// TIA Portal V18 export
// export: Created 2025-12-01T17:50:25.5329031Z, ExportSetting None, DisplayName Totally Integrated Automation Portal, DisplayVersion V18 Update 5, DisplayName TIA Portal Openness, DisplayVersion V18 Update 5, DisplayName TIA Portal Teamcenter Gateway, DisplayVersion V18, DisplayName TIA Portal Version Control Interface, DisplayVersion V18, DisplayName STEP 7 Professional, DisplayVersion V18 Update 5, DisplayName STEP 7 Safety, DisplayVersion V18, DisplayName WinCC Professional, DisplayVersion V18 Update 5
ORGANIZATION_BLOCK "07_CYCL_FLT"   // OB80, STL, TimeErrorInterrupt
TITLE = "Cycle Time Fault"
{ S7_Optimized_Access := 'FALSE' }
   VAR_TEMP
      OB80_EV_CLASS : Byte;   // 16#35, Event class 3, Entering event state, Internal fault event
      OB80_FLT_ID : Byte;   // 16#XX, Fault identifcation code
      OB80_PRIORITY : Byte;   // Priority of OB Execution
      OB80_OB_NUMBR : Byte;   // 80 (Organization block 80, OB80)
      OB80_RESERVED_1 : Byte;   // Reserved for system
      OB80_RESERVED_2 : Byte;   // Reserved for system
      OB80_ERROR_INFO : Word;   // Error information on event
      OB80_ERR_EV_CLASS : Byte;   // Class of event causing error
      OB80_ERR_EV_NUM : Byte;   // Number of event causing error
      OB80_OB_PRIORITY : Byte;   // Priority of OB causing error
      OB80_OB_NUM : Byte;   // Number of OB causing error
      OB80_DATE_TIME : Date_And_Time;   // Date and time OB80 started
   END_VAR
BEGIN
END_ORGANIZATION_BLOCK
